# EPICS substitutions: Epics_Installation/gpib_test/gpib_test/gpibApp/Db/Keithley6485.substitutions
file Keithley6485Main.template {
pattern { PROTO }
    { Keithley6485.proto }
}

file SCPI.template {
pattern { PROTO }
    { Keithley6485.proto }
}
